FUNCTION_BLOCK AOI_DeltaScaraRobot
VAR_INPUT
END_VAR
VAR_OUTPUT
END_VAR
VAR
	rtStart: R_trig;
	rtStop: R_Trig;
	rtHold: R_Trig;
END_VAR
VAR_IN_OUT
	Scara: UDT_Scara;
END_VAR

IF Scara.i.Auto THEN
   Scara.Di_[1][4]:=0;
   Scara.Di_[1][5]:=1;   
   ELSE IF Scara.i.T2  THEN
	      Scara.Di_[1][4]:=1;
          Scara.Di_[1][5]:=1;     
         END_IF 		
END_IF

IF rtStart.Q  THEN
   Scara.Di_[1][6]:=1;
   Scara.Di_[1][7]:=1;
END_IF   
IF Scara.i.Stop THEN
   Scara.Di_[1][6]:=1;
   Scara.Di_[1][7]:=0;
END_IF   
IF rtHold.Q THEN
	Scara.Di_[1][6]:=0;
	Scara.Di_[1][7]:=1;
END_IF


rtStart(CLK:=Scara.i.Start , Q=> );
rtStop(CLK:=Scara.i.Stop , Q=> );
rtHold(CLK:=Scara.i.Hold , Q=> );

Scara.Di_[1][1]:=NOT Scara.i.Estop AND NOT Scara.i.Shutdown ;
Scara.Di_[1][2]:=NOT Scara.i.Estop;
Scara.Di_[1][3]:=Scara.i.Reset;
Scara.Di_[1][8]:=Scara.i.reset OR scara.i.FuctionReset;

Scara.o.Error:=Scara.Do_[1][1];
Scara.o.Enable:=Scara.Do_[1][2];
Scara.o.InPos:=Scara.Do_[1][3];
Scara.o.FuctionHold:=Scara.Do_[1][4];
Scara.o.ProRunning:=Scara.Do_[1][5] AND Scara.Do_[1][6];
Scara.o.Held:=NOT Scara.Do_[1][5] AND Scara.Do_[1][6];
Scara.o.ProStopped:= Scara.Do_[1][5] AND NOT Scara.Do_[1][6];

Scara.Di_[2][1]:=Scara.i.ProFaultClear;
Scara.Di_[2][2]:=Scara.i.ProPick;
Scara.Di_[2][3]:=Scara.i.ProDepart;
Scara.Di_[2][4]:=Scara.i.ProPut;
Scara.Di_[2][5]:=Scara.i.LoopStop;//循环停止

Scara.o.ProFault:=Scara.Do_[2][1];
Scara.o.ProPickDone:=Scara.Do_[2][2];
Scara.o.ProPutDone:=Scara.Do_[2][3];
Scara.o.ProDepartDone:=Scara.Do_[2][4];
Scara.o.LoopStopDone:=Scara.Do_[2][5];//循环完成
Scara.o.ResettingDone:=Scara.Do_[2][6];//复位完成

END_FUNCTION_BLOCK

(* stored: Version 1.1.0.1, ProductVersion 3.1.4022.16
   POU AOI_DeltaScaraRobot: Id {7ccf4f04-80f1-47ce-82b8-5de0d8cc1692}, SpecialFunc None *)
